TYPE MySecondStructure :
STRUCT
	myLint : LINT;
	myDint : DINT;
END_STRUCT
END_TYPE

(* stored: Version 1.1.0.1, ProductVersion 3.1.4024.11
   DUT MySecondStructure: Id {903da5a0-ff7a-4726-8ba5-7896a90f4738} *)
